(* CoDeSys 2.3.9.22 project: pk1.pro *)
(* Libraries: STANDARD.LIB 4.10.05 11:14:46, IECSFC.LIB 13.4.06 15:51:28, ANALYZATION.LIB 5.10.99 09:05:06 *)

(* PLC configuration (modules and I/O channels)
start AT %IX0.0 [BitInput]
stop AT %IX0.1 [BitInput]
avar AT %IX0.2 [BitInput]
AT %IX0.3 [BitInput]
AT %IX0.4 [BitInput]
AT %IX0.5 [BitInput]
Discrete output 4 bit [ID101] node 1, in %IB1 out %QB1 {PinCount = 4; SafeValueBool = FALSE; SafeValueBool = FALSE; SafeValueBool = FALSE; SafeValueBool = FALSE; Visibility = No}
  AT %QX1.0 [BitOutput]
  AT %QX1.1 [BitOutput]
  AT %QX1.2 [BitOutput]
  AT %QX1.3 [BitOutput]
Special output [ID104] node 2, in %IB2 out %QB2 {Visibility = No; PinCount = 1}
  AT %QX2.0 [BitOutput] Special output
Unifed signal sensor [ID700] node 3, in %IB3 out %QB3 {Type_of_sensor700 = IT_0_20; measure_interval = 0.8; ainlow = 0; ainhigh = 20; first_cor_point = 0; first_delta = 0; second_cor_point = 0; second_delta = 0; third_cor_point = 0; third_delta = 0; Visibility = No}
  AT %ID3.0 [FloatInput] Value
  AT %IW3.1 [WordInput] Circular time
  Analog Input [ID107] node 0, in %IB3.0 out %QB3.0
Unifed signal sensor [ID700] node 4, in %IB4 out %QB4 {Type_of_sensor700 = IT_0_20; measure_interval = 0.8; ainlow = 0; ainhigh = 20; first_cor_point = 0; first_delta = 0; second_cor_point = 0; second_delta = 0; third_cor_point = 0; third_delta = 0; Visibility = No}
  AT %ID4.0 [FloatInput] Value
  AT %IW4.1 [WordInput] Circular time
  Analog Input [ID107] node 0, in %IB4.0 out %QB4.0
Unifed signal sensor [ID700] node 5, in %IB5 out %QB5 {Type_of_sensor700 = IT_0_20; measure_interval = 0.8; ainlow = 0; ainhigh = 20; first_cor_point = 0; first_delta = 0; second_cor_point = 0; second_delta = 0; third_cor_point = 0; third_delta = 0; Visibility = No}
  AT %ID5.0 [FloatInput] Value
  AT %IW5.1 [WordInput] Circular time
  Analog Input [ID107] node 0, in %IB5.0 out %QB5.0
Unifed signal sensor [ID700] node 6, in %IB6 out %QB6 {Type_of_sensor700 = IT_0_20; measure_interval = 0.8; ainlow = 0; ainhigh = 20; first_cor_point = 0; first_delta = 0; second_cor_point = 0; second_delta = 0; third_cor_point = 0; third_delta = 0; Visibility = No}
  AT %ID6.0 [FloatInput] Value
  AT %IW6.1 [WordInput] Circular time
  Analog Input [ID107] node 0, in %IB6.0 out %QB6.0
Analog output [ID106] node 7, in %IB7 out %QB7 {DAC_Type = Current 4-20mA; Analog_offset_correction = 0; Analog_full_range_correction = 0; SafeValueFloat = 0; Visibility = No}
  AT %QD7.0 [FloatOutput] Value
Analog output [ID106] node 8, in %IB8 out %QB8 {DAC_Type = Current 4-20mA; Analog_offset_correction = 0; Analog_full_range_correction = 0; SafeValueFloat = 0; Visibility = No}
  AT %QD8.0 [FloatOutput] Value
*)

(* POU PLC_PRG, CFC *)
PROGRAM PLC_PRG
VAR
	rs1: RS;
	ctu1: CTU;
	x: REAL;
	ton1: TON;
	etX1: REAL;
	etY1: REAL;
	ton2: TON;
	ton3: TON;
	etX2: REAL;
	ton4: TON;
	rs2: RS;
	k5: BOOL;
	k4: BOOL;
	k1: BOOL;
	k3: BOOL;
	on: BOOL;
	off: BOOL;
	tp1: TP;
END_VAR
VAR (* helpers for the ST form of the networks *)
	_t126 : BOOL;
END_VAR
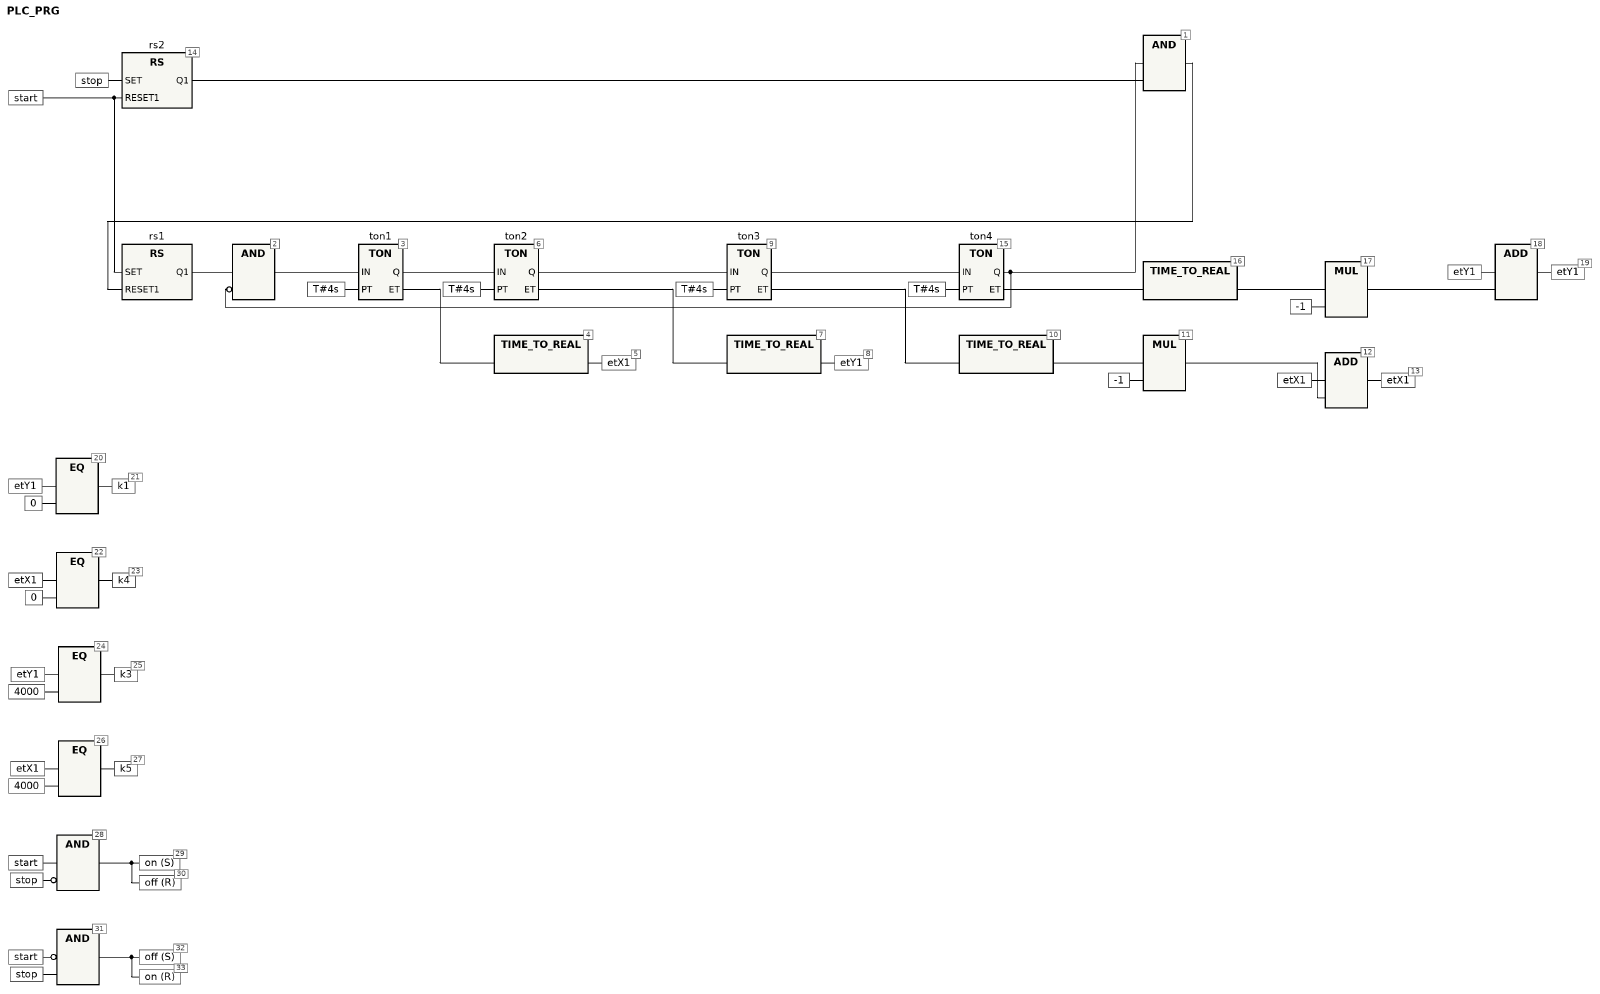
_CFC_ (* Continuous Function Chart, elements in execution order *)
#0 rs1:RS(SET: start, RESET1: #1)
#1 AND(#15.Q, #14.Q1)
#2 AND(#0.Q1, NOT #15.Q)
#3 ton1:TON(IN: #2, PT: T#4s)
#4 TIME_TO_REAL(#3.ET)
#5 etX1 <= #4
#6 ton2:TON(IN: #3.Q, PT: T#4s)
#7 TIME_TO_REAL(#6.ET)
#8 etY1 <= #7
#9 ton3:TON(IN: #6.Q, PT: T#4s)
#10 TIME_TO_REAL(#9.ET)
#11 MUL(#10, -1)
#12 ADD(etX1, #11)
#13 etX1 <= #12
#14 rs2:RS(SET: stop, RESET1: start)
#15 ton4:TON(IN: #9.Q, PT: T#4s)
#16 TIME_TO_REAL(#15.ET)
#17 MUL(#16, -1)
#18 ADD(etY1, #17)
#19 etY1 <= #18
#20 EQ(etY1, 0)
#21 k1 <= #20
#22 EQ(etX1, 0)
#23 k4 <= #22
#24 EQ(etY1, 4000)
#25 k3 <= #24
#26 EQ(etX1, 4000)
#27 k5 <= #26
#28 AND(start, NOT stop)
#29 S on <= #28
#30 R off <= #28
#31 AND(NOT start, stop)
#32 S off <= #31
#33 R on <= #31
_END_CFC_
(* the same logic as Structured Text *)
rs1(SET := start, RESET1 := _t126);
_t126 := ton4.Q AND rs2.Q1;
ton1(IN := rs1.Q1 AND NOT ton4.Q, PT := T#4s);
etX1 := TIME_TO_REAL(ton1.ET);
ton2(IN := ton1.Q, PT := T#4s);
etY1 := TIME_TO_REAL(ton2.ET);
ton3(IN := ton2.Q, PT := T#4s);
etX1 := etX1 + (TIME_TO_REAL(ton3.ET) * (-1));
rs2(SET := stop, RESET1 := start);
ton4(IN := ton3.Q, PT := T#4s);
etY1 := etY1 + (TIME_TO_REAL(ton4.ET) * (-1));
k1 := etY1 = 0;
k4 := etX1 = 0;
k3 := etY1 = 4000;
k5 := etX1 = 4000;
IF start AND NOT stop THEN on := TRUE; END_IF;
IF start AND NOT stop THEN off := FALSE; END_IF;
IF NOT start AND stop THEN off := TRUE; END_IF;
IF NOT start AND stop THEN on := FALSE; END_IF;
END_PROGRAM

(* Visualisation viz
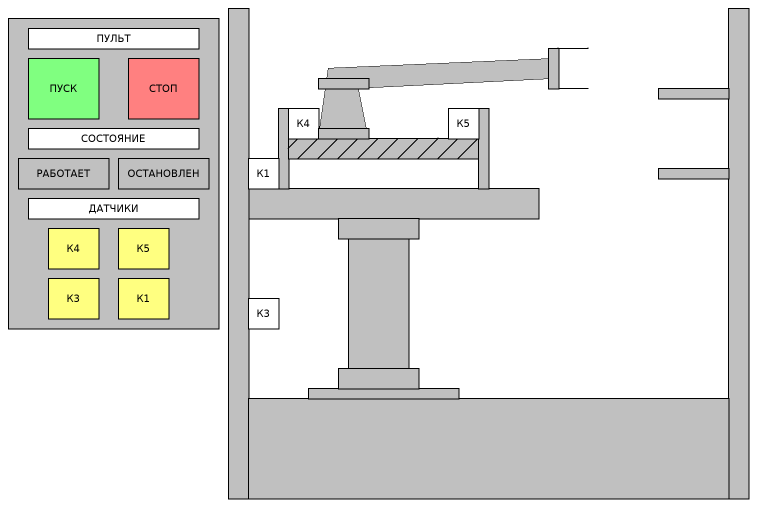
rounded rectangle at (30,60)-(101,121): text "ПУСК"; alarm colour if .start; taps .start
rounded rectangle at (130,60)-(201,121): text "СТОП"; alarm colour if .stop; taps .stop
polygon at (310,60)-(560,140): x offset PLC_PRG.etX1/50; y offset PLC_PRG.etY1/50
rectangle at (250,300)-(281,331): text "К3"; alarm colour if PLC_PRG.k3
rectangle at (250,160)-(281,191): text "К1"; alarm colour if PLC_PRG.k1
rectangle at (450,110)-(481,141): text "К5"; alarm colour if PLC_PRG.k5; y offset PLC_PRG.etY1/50
rectangle at (290,110)-(321,141): text "К4"; alarm colour if PLC_PRG.k4; y offset PLC_PRG.etY1/50
polyline at (560,50)-(590,60): x offset PLC_PRG.etX1/50; y offset PLC_PRG.etY1/50
polyline at (560,80)-(590,90): x offset PLC_PRG.etX1/50; y offset PLC_PRG.etY1/50
rounded rectangle at (320,130)-(371,141): x offset PLC_PRG.etX1/50; y offset PLC_PRG.etY1/50
rounded rectangle at (320,80)-(371,91): x offset PLC_PRG.etX1/50; y offset PLC_PRG.etY1/50
rounded rectangle at (550,50)-(561,91): x offset PLC_PRG.etX1/50; y offset PLC_PRG.etY1/50
rectangle at (30,30)-(201,51): text "ПУЛЬТ"
rectangle at (30,200)-(201,221): text "ДАТЧИКИ"
rounded rectangle at (50,230)-(101,271): text "К4"; alarm colour if PLC_PRG.k4
rounded rectangle at (120,230)-(171,271): text "К5"; alarm colour if PLC_PRG.k5
rounded rectangle at (120,280)-(171,321): text "К1"; alarm colour if PLC_PRG.k1
rounded rectangle at (50,280)-(101,321): text "К3"; alarm colour if PLC_PRG.k3
rectangle at (30,130)-(201,151): text "СОСТОЯНИЕ"
rounded rectangle at (120,160)-(211,191): text "ОСТАНОВЛЕН"; alarm colour if PLC_PRG.off
rounded rectangle at (20,160)-(111,191): text "РАБОТАЕТ"; alarm colour if PLC_PRG.on
24 more shapes without text or variables
*)
